// SIMATIC S7-200 SMART project (STEP 7-Micro/WIN SMART), CPU SR20

SYMBOL_TABLE System Symbols
Always_On        SM0.0    // Always ON
First_Scan_On    SM0.1    // ON for the first scan cycle only
HSC0_Ctrl        SMB37    // Configure and control HSC0
HSC0_CV          SMD38    // HSC0 new current value
HSC0_PV          SMD42    // HSC0 new preset value
END_SYMBOL_TABLE

ORGANIZATION_BLOCK MAIN:OB1
TITLE=Program Comments
BEGIN
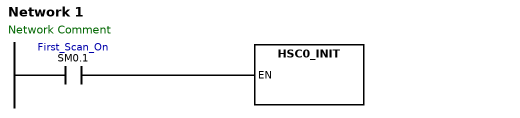
Network 1
// Network Comment
LD     First_Scan_On:SM0.1
CALL   HSC0_INIT:SBR1
END_ORGANIZATION_BLOCK

SUBROUTINE_BLOCK HSC0_INIT:SBR1
TITLE=
BEGIN
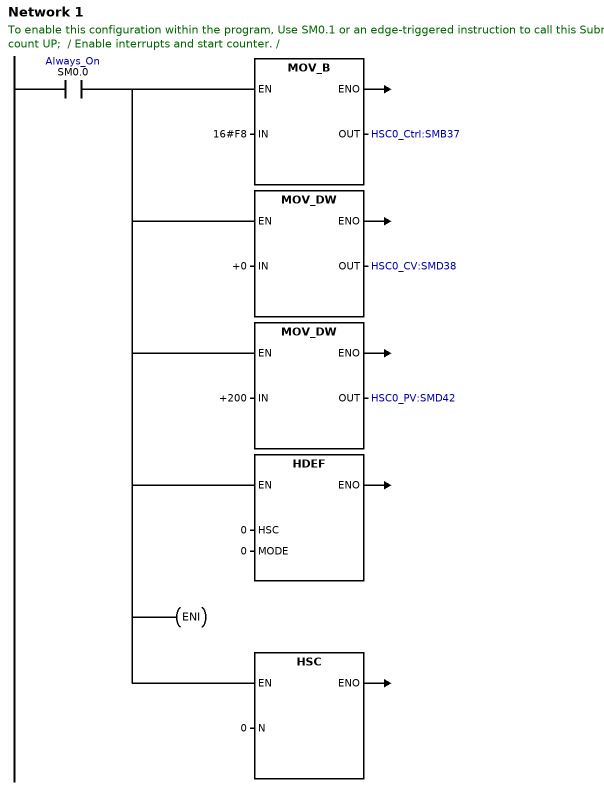
Network 1
// To enable this configuration within the program, Use SM0.1 or an edge-triggered instruction to call this Subroutine once from the MAIN program block.  
// Configure HC0 for Mode 0; CV = 0; PV = 200; count UP; 
// Enable interrupts and start counter.
// 
//Set control bits: count UP; enabled; 
//Load CV
//Load PV
LD     Always_On:SM0.0
MOVB   16#F8, HSC0_Ctrl:SMB37
MOVD   +0, HSC0_CV:SMD38
MOVD   +200, HSC0_PV:SMD42
HDEF   0, 0
ENI
HSC    0
END_SUBROUTINE_BLOCK
